// Mitsubishi GX Works2 project: 20240318_AI机程序新增MODBUS-通道2   PLC: FX3S

PROGRAM MAIN
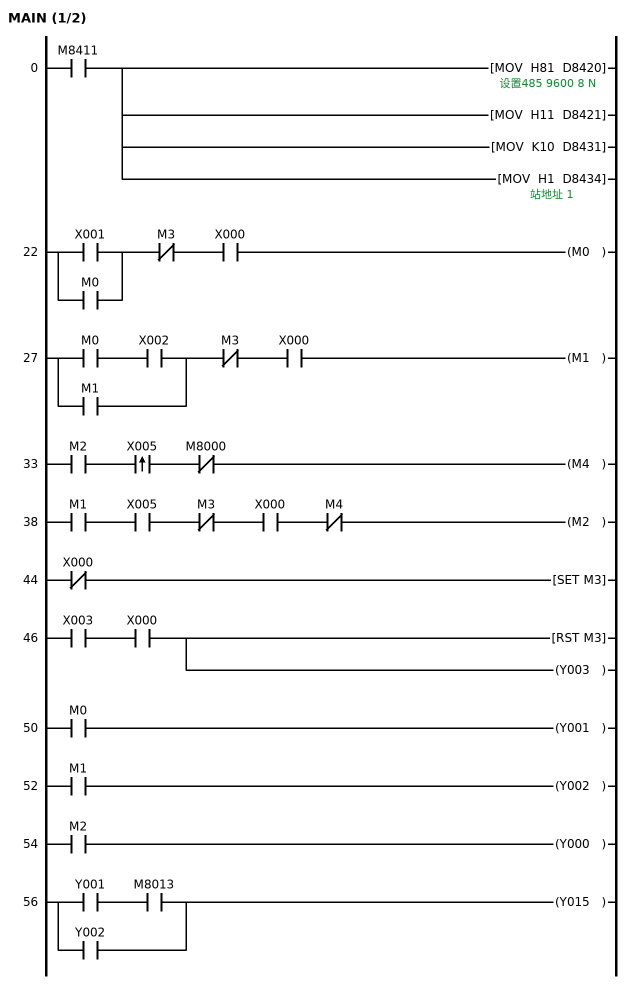
0     LD      M8411
      MOV     H81 D8420  ; 设置485 9600 8 N
      MOV     H11 D8421
      MOV     K10 D8431
      MOV     H1 D8434  ; 站地址 1
22    LD      X001
      OR      M0
      ANI     M3
      AND     X000
      OUT     M0
27    LD      M0
      AND     X002
      OR      M1
      ANI     M3
      AND     X000
      OUT     M1
33    LD      M2
      ANDP    X005
      ANI     M8000
      OUT     M4
38    LD      M1
      AND     X005
      ANI     M3
      AND     X000
      ANI     M4
      OUT     M2
44    LDI     X000
      SET     M3
46    LD      X003
      AND     X000
      RST     M3
      OUT     Y003
50    LD      M0
      OUT     Y001
52    LD      M1
      OUT     Y002
54    LD      M2
      OUT     Y000
56    LD      Y001
      AND     M8013
      OR      Y002
      OUT     Y015
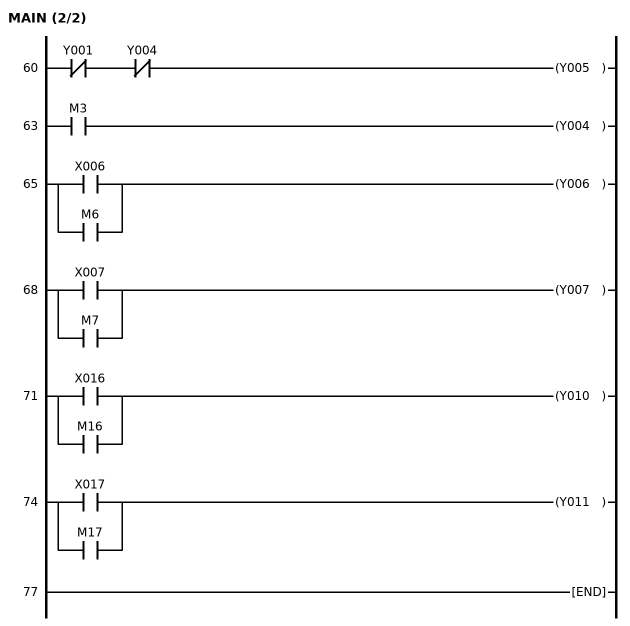
60    LDI     Y001
      ANI     Y004
      OUT     Y005
63    LD      M3
      OUT     Y004
65    LD      X006
      OR      M6
      OUT     Y006
68    LD      X007
      OR      M7
      OUT     Y007
71    LD      X016
      OR      M16
      OUT     Y010
74    LD      X017
      OR      M17
      OUT     Y011
77    END
END_PROGRAM
